# EPICS IOC start-up script: iocBoot/iocCITests/testLInt.iocsh
#!../../bin/linux-x86_64/omroneipApp
< envPaths
epicsEnvSet("P", "omronEIP:")
epicsEnvSet("EPICS_CAS_INTF_ADDR_LIST", "127.0.0.1")
epicsEnvSet("EPICS_CA_ADDR_LIST", "127.0.0.1")

cd ${TOP}
dbLoadDatabase("dbd/omroneipApp.dbd")
omroneipApp_registerRecordDeviceDriver(pdbbase)

#drvOmronEIPConfigure(driverPortName, gateway, route_path, plc, libplctag_debug)
drvOmronEIPConfigure("omronDriver", "127.0.0.1", "${PLC_GATEWAY}", "${PLC}", 1, 0)

#drvOmronEIPConfigPoller(driverPortName, pollerName, updateRate, spreadRequests)
drvOmronEIPConfigPoller("omronDriver", "fastPoller", 1, 1) #This can be lowered to 0.1

dbLoadRecords("db/CI_testLInt.db", "P=${P}, PORT=omronDriver, POLLER=fastPoller")

iocInit()

dbl()
